Universal Robots PolyScope program: Triangle.urp

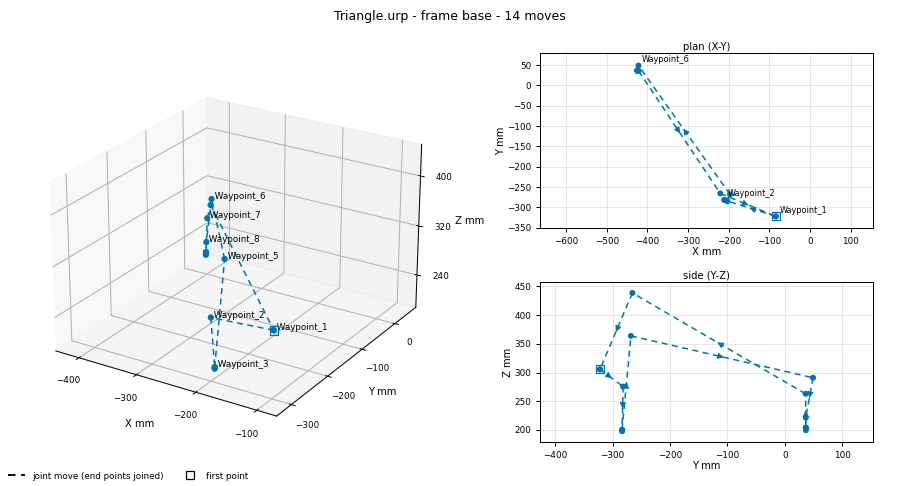
[picture p0: tool path of Triangle.urp in frame base, 14 of 14 moves have a stored position in this frame; points joined in program order, loops and branches not executed]
Program Triangle (installation=default directory=/programs/usbdisk/Zahra1 createdIn=5.11.11.1010533 lastSavedIn=5.11.11.1010533 robotSerialNumber=20205300864)
Calibrated DH parameters: a=[-0.000166, -0.243494, -0.153108, 0.000057, -0.000123, 0]; d=[0.151897, -1.34267, 53.988124, -52.514559, 0.085283, 0.092193]; alpha=[1.572472, -0.003756, 0.002824, 1.570807, -1.572621, 0]; deltaTheta=[0, 0.020704, 7.033215, -0.770746, 0.000004, 0]
Robot Program (runOnlyOnce=true)
  MoveJ speed 60 deg/s, acceleration 80 deg/s^2 (useActiveTCP=true) feature=Base
    Waypoint Waypoint_1: TCP in base x=-84.297 y=-321.869 z=305.472 mm, rx=-2.081 ry=-2.2572 rz=0.0983 rad; joints [-79.978, -91.2, -87.974, -91.699, 84.673, 815.507] deg
    Waypoint Waypoint_2: TCP in base x=-211.336 y=-281.592 z=275.53 mm, rx=-2.2116 ry=-2.1482 rz=0.0226 rad; joints [-104.227, -96.89, -89.784, -84.266, 86.727, 797.577] deg
    Waypoint Waypoint_3: TCP in base x=-204.211 y=-283.39 z=200.204 mm, rx=-2.258 ry=-2.1295 rz=0.0363 rad; joints [-103.17, -101.313, -106.185, -62.479, 87.485, 800.347] deg
    Waypoint Waypoint_4: TCP in base x=-204.289 y=-283.374 z=197.862 mm, rx=-2.2579 ry=-2.1296 rz=0.0361 rad; joints [-103.186, -101.589, -106.546, -61.845, 87.489, 800.329] deg
    URCap Gripper (Robotiq_Grippers, Robotiq Inc.) dataModel(position=70.98039215686275, force=97.0, speed=52.0, positionInDouble=70.98039215686275, forceInDouble=97.0, speedInDouble=52.0, slaveIds=[9], blocking=true, robotCompliant=false)
    Waypoint Waypoint_3: motionParameters(jointSpeed=0.698132 jointAcceleration=0.349066 cartesianSpeed=0.25 cartesianAcceleration=1.2); TCP in base x=-204.211 y=-283.39 z=200.204 mm, rx=-2.258 ry=-2.1295 rz=0.0363 rad; joints [-103.17, -101.313, -106.185, -62.479, 87.485, 800.347] deg
    Waypoint Waypoint_5: TCP in base x=-196.923 y=-267.941 z=363.759 mm, rx=-1.9785 ry=-2.388 rz=0.1084 rad; joints [-102.036, -91.889, -72.78, -102.702, 86.166, 787.233] deg
    Waypoint Waypoint_6: TCP in base x=-422.067 y=48.996 z=290.864 mm, rx=-1.4524 ry=-2.7169 rz=0.0697 rad; joints [-168.694, -113.955, -65.543, -86.093, 89.746, 697.635] deg
    Waypoint Waypoint_8: TCP in base x=-424.022 y=36.35 z=221.802 mm, rx=-1.6263 ry=-2.6315 rz=0.0332 rad; joints [-166.832, -116.819, -79.415, -70.849, 88.883, 706.687] deg
    Waypoint Waypoint_9: TCP in base x=-424.953 y=36.463 z=204.094 mm, rx=-1.6263 ry=-2.6314 rz=0.0334 rad; joints [-166.885, -118.366, -82.02, -66.689, 88.885, 706.644] deg
    Waypoint Waypoint_10: motionParameters(jointSpeed=0.698132 jointAcceleration=0.349066 cartesianSpeed=0.25 cartesianAcceleration=1.2); TCP in base x=-425.18 y=36.491 z=199.655 mm, rx=-1.6263 ry=-2.6315 rz=0.0333 rad; joints [-166.899, -118.796, -82.611, -65.672, 88.888, 706.632] deg
    URCap Gripper (Robotiq_Grippers, Robotiq Inc.) dataModel(position=40.3921568627451, force=97.0, speed=52.0, positionInDouble=40.3921568627451, forceInDouble=97.0, speedInDouble=52.0, slaveIds=[9], blocking=true, robotCompliant=false)
    Waypoint Waypoint_9: TCP in base x=-424.953 y=36.463 z=204.094 mm, rx=-1.6263 ry=-2.6314 rz=0.0334 rad; joints [-166.885, -118.366, -82.02, -66.689, 88.885, 706.644] deg
    Waypoint Waypoint_7: TCP in base x=-421.866 y=36.066 z=263.013 mm, rx=-1.6263 ry=-2.6314 rz=0.0334 rad; joints [-166.704, -114.326, -71.866, -80.885, 88.869, 706.799] deg
    Waypoint Waypoint_12: TCP in base x=-220.963 y=-265.49 z=438.519 mm, rx=-0.9439 ry=-2.8214 rz=0.1399 rad; joints [-104.67, -102.553, -39.092, -123.473, 80.196, 741.944] deg
    Waypoint Waypoint_1: TCP in base x=-84.297 y=-321.869 z=305.472 mm, rx=-2.081 ry=-2.2572 rz=0.0983 rad; joints [-79.978, -91.2, -87.974, -91.699, 84.673, 815.507] deg
